// SIMATIC S7-200 project (STEP 7-Micro/WIN), CPU 221 REL 01.10

ORGANIZATION_BLOCK MAIN:OB1
TITLE=The elevator control system triggers corresponding actions through external and internal call buttons across various logic segments. When an employee presses an external call button for a specific floor, the system determines whether to illuminate the corresponding external call response light based on the position sensor. If movement to the target floor is required, the system activates either the upward or downward motor control, ensuring they do not operate simultaneously; the running indicator light is separately illuminated to signal elevator operation.
// Upon reaching the target floor, the system activates the door open control, with a delay timer maintaining the open duration; the door open control for a specific floor is only activated if the door is not already open, preventing redundant opening. When passengers select an internal call button, the system illuminates the corresponding response light, and the door close control is separately initiated to close the elevator door.
// Safety mechanisms are paramount. The overload sensor triggers the overload indicator light, and motor controls are separately halted. If the emergency stop button is pressed, the emergency stop indicator light illuminates, and a delay timer later resets the call button lock. In case of a fault, the fault indicator light illuminates, and the alarm is separately activated; internal lighting is simultaneously turned on to provide illumination for passengers.
// The external call response light illuminates upon confirmation from the position sensor, requiring cooperation from the external call button. The door open control is coordinated via a delay timer, with the door close control operating separately to ensure smooth door operation.
BEGIN
Network 1 // NETWORK TITLE (single line)
//  
// NETWORK COMMENTS
//  
// 
LD     I0.0
O      Q0.0
O      I0.5
O      M1.1
O      I0.4
AN     I0.2
AN     Q0.1
=      Q0.0
Network 2
LD     I0.1
O      Q0.1
O      T37
AN     I0.0
AN     I0.5
AN     I0.3
AN     I0.4
AN     Q0.0
=      Q0.1
Network 3
LD     I0.2
O      M0.0
AN     T37
=      M0.0
A      M0.1
TON    T37, +20
Network 4
LD     Q0.0
O      Q0.1
TON    T38, +5
AN     T38
=      Q0.2
Network 5
LD     I2.0
O      Q0.6
AN     M0.3
=      Q0.6
ED
=      M2.0
Network 6
LD     I2.1
O      Q0.7
AN     M0.4
=      Q0.7
ED
=      M2.1
Network 7
LD     I2.2
O      Q1.0
AN     M0.5
=      Q1.0
ED
=      M2.2
Network 8
LD     I2.3
O      Q1.1
AN     M0.6
=      Q1.1
ED
=      M2.3
Network 9
LD     I0.6
O      Q2.0
LDN    M0.3
O      M1.0
ALD
=      Q2.0
ED
=      M2.4
Network 10
LD     I0.7
O      Q2.1
LDN    M0.4
O      M1.0
ALD
=      Q2.1
ED
=      M2.5
Network 11
LD     I1.0
O      Q2.2
LDN    M0.5
O      M1.0
ALD
=      Q2.2
ED
=      M2.6
Network 12
LD     I1.1
O      Q2.3
LDN    M0.4
O      M0.7
ALD
=      Q2.3
ED
=      M2.7
Network 13
LD     I1.2
O      Q2.4
LDN    M0.5
O      M0.7
ALD
=      Q2.4
ED
=      M3.0
Network 14
LD     I1.3
O      Q2.5
LDN    M0.6
O      M0.7
ALD
=      Q2.5
ED
=      M3.1
Network 15
LD     Q0.6
O      Q0.7
O      Q1.0
O      Q1.1
=      M0.1
Network 16
LD     Q2.0
O      Q2.1
O      Q2.2
O      Q2.3
O      Q2.4
O      Q2.5
=      M0.2
Network 17
LD     I2.6
A      I2.7
=      M0.3
Network 18
LD     I3.0
A      I3.1
=      M0.4
Network 19
LD     I3.2
A      I3.3
=      M0.5
Network 20
LD     I3.4
A      I3.5
=      M0.6
Network 21
LD     I2.6
O      I2.7
O      Q3.0
AN     I3.0
AN     Q3.1
AN     Q3.2
AN     Q3.3
=      Q3.0
Network 22
LD     I3.0
O      I3.1
O      Q3.1
AN     I2.7
AN     I3.2
AN     Q3.0
AN     Q3.2
AN     Q3.3
=      Q3.1
Network 23
LD     I3.2
O      I3.3
O      Q3.2
AN     I3.1
AN     I3.4
AN     Q3.0
AN     Q3.1
AN     Q3.3
=      Q3.2
Network 24
LD     I3.4
O      I3.5
O      Q3.3
AN     I3.3
AN     Q3.0
AN     Q3.1
AN     Q3.2
=      Q3.3
Network 25
LD     Q0.7
AN     M0.4
O      Q1.0
AN     M0.5
O      Q1.1
AN     M0.6
AN     M1.0
=      M0.7
=      Q2.6
Network 26
LD     Q1.0
AN     M0.5
O      Q0.7
AN     M0.4
O      Q0.6
AN     M0.3
AN     M0.7
=      M1.0
=      Q2.7
Network 27
LD     M0.7
AN     I3.7
A      I0.3
AN     I3.6
AN     M1.1
AN     T40
AN     Q0.4
=      Q0.3
Network 28
LD     M1.0
AN     I3.7
A      I0.3
AN     I2.5
AN     M1.1
AN     T40
AN     Q0.3
=      Q0.4
Network 29
LD     I2.6
O      I2.7
A      Q0.6
LD     Q2.1
A      M0.7
LD     Q2.3
A      M1.0
OLD
O      Q0.7
LD     I3.0
O      I3.1
ALD
OLD
LD     Q2.2
A      M0.7
LD     Q2.4
A      M1.0
OLD
O      Q1.0
LD     I3.2
O      I3.3
ALD
OLD
LD     I3.4
O      I3.5
A      Q1.1
OLD
=      M1.2
Network 30
LD     M0.7
O      M1.0
AN     M1.2
=      Q0.5
Network 31
LD     M2.0
O      M2.1
O      M2.2
O      M2.3
O      M2.4
O      M2.5
O      M2.6
O      M2.7
O      M3.0
O      M3.1
=      M1.1
Network 32
LD     M1.1
TOF    T40, +10
Network 33
LD     M1.1
O      Q3.6
AN     T39
=      Q3.6
TON    T39, +10
END_ORGANIZATION_BLOCK
